Staubli VAL3: putButton.pgx

public program putButton(num nValue, string sText)
begin
  // Puts a text label above a function key
  //
  // Labels greater than 4 characters will shorten to 4
  //
  // copyright (c) 2015-2021 victortorreslopez
  //
  // GNU General Public License
  //
  // Parameters
  // - nValue: number of function key (1..8)
  // - sText: function key label
  //
  // References
  // - "2005-27 Example Application". Staubli. 2005
  //
  // Version history
  // ---------------
  // 0.1, 2021/12/21, VTL: centers the label
  // 0.0, 2015/01/14, VTL: alfa release

  if (nValue >= 1) and (nValue <= 8)
    if (len(sText) > 4)
      sText = left(sText, 3) + "."
    endIf
    gotoxy(((nValue - 1) * 5) + round((5 - len(sText)) / 2), 13)
    put(sText)
  endIf
end
